PROGRAM MAIN
VAR
	MainReadIO : StReadIO;
	FB_SystemTest : SystemTest;
END_VAR

FB_SystemTest();

MainReadIO.st_ReadIO := IO.g_ReadIO;

END_PROGRAM

(* stored: Version 1.1.0.1, ProductVersion 3.1.4024.6
   POU MAIN: Id {e10f5808-78da-4366-9b27-b0c1d74ac72a}, SpecialFunc None *)
